KUKA KRL program: CONCERT.src, CONCERT.dat

--- CONCERT.src ---
&ACCESS RVO
&REL 519
&PARAM EDITMASK = *
&PARAM TEMPLATE = C:\KRC\Roboter\Template\vorgabe
&PARAM DISKPATH = KRC:\R1\Program\_KLAVIRISTA_V2\subprogram
DEF CONCERT( )
;FOLD INI
CONTINUE
IF NOT $ON_PATH THEN
  ;FOLD BASISTECH INI
    GLOBAL INTERRUPT DECL 3 WHEN $STOPMESS==TRUE DO IR_STOPM ( )
    INTERRUPT ON 3
    BAS (#INITMOV,0 )
  ;ENDFOLD (BASISTECH INI)
  ;FOLD USER INI
    ;Make your modifications here

  ;ENDFOLD (USER INI)
ENDIF
  ;ENDFOLD (INI)
;FOLD PTP HOME1 Vel=8 % PDAT5 ;%{PE}
;FOLD Parameters ;%{h}
;Params IlfProvider=kukaroboter.basistech.inlineforms.movement.old; Kuka.IsGlobalPoint=False; Kuka.PointName=HOME1; Kuka.BlendingEnabled=False; Kuka.MoveDataPtpName=PDAT5; Kuka.VelocityPtp=100; Kuka.CurrentCDSetIndex=0; Kuka.MovementParameterFieldEnabled=True; IlfCommand=PTP
;ENDFOLD
$BWDSTART = FALSE
PDAT_ACT = PPDAT5
FDAT_ACT = FHOME1
BAS(#PTP_PARAMS, 8)
SET_CD_PARAMS (0)
PTP XHOME1
;ENDFOLD

;FOLD PTP HOME1 Vel=8 % PDAT5 ;%{PE}
;FOLD Parameters ;%{h}
;Params IlfProvider=kukaroboter.basistech.inlineforms.movement.old; Kuka.IsGlobalPoint=False; Kuka.PointName=HOME1; Kuka.BlendingEnabled=False; Kuka.MoveDataPtpName=PDAT5; Kuka.VelocityPtp=100; Kuka.CurrentCDSetIndex=0; Kuka.MovementParameterFieldEnabled=True; IlfCommand=PTP
;ENDFOLD
$BWDSTART = FALSE
PDAT_ACT = PPDAT5
FDAT_ACT = FHOME1
BAS(#PTP_PARAMS, 8)
SET_CD_PARAMS (0)
PTP XHOME1
;ENDFOLD

END
GLOBAL DEF PLAY(KEY:IN, TIME:IN, HOLD:IN)
;FOLD Variables INI
REAL KEY
INT TIME
INT HOLD
INT PRESS
INT SPEED
REAL SHIFT
;ENDFOLD
PRESS = 10
SHIFT = 23.3
SPEED = 17
$TIMER_STOP[1]=FALSE
;FOLD STATUS TREATMENT
KEY = KEY+7
IF KEY < 11 THEN
XP1 = START4
ELSE
XP1 = START5
ENDIF
;IF KEY <= 8 THEN
;XP1 = START1
;ENDIF
;IF (KEY > 8) AND (KEY < 11) THEN
;XP1 = START2
;ENDIF
;IF KEY >= 11 THEN
;XP1 = START3
;ENDIF
;ENDFOLD

XP1.X = XP1.X + (KEY-1) * SHIFT
;FOLD PTP P1 Vel=100 % PDAT1 Tool[4]:TQGripper Base[1]:Piano ;%{PE}
;FOLD Parameters ;%{h}
;Params IlfProvider=kukaroboter.basistech.inlineforms.movement.old; Kuka.IsGlobalPoint=False; Kuka.PointName=P1; Kuka.BlendingEnabled=False; Kuka.MoveDataPtpName=PDAT1; Kuka.VelocityPtp=100; Kuka.CurrentCDSetIndex=0; Kuka.MovementParameterFieldEnabled=True; IlfCommand=PTP
;ENDFOLD
$BWDSTART = FALSE
PDAT_ACT = PPDAT1
FDAT_ACT = FP1
BAS(#PTP_PARAMS, SPEED)
SET_CD_PARAMS (0)
PTP XP1
;ENDFOLD
XP1.Z = XP1.Z - PRESS
WAIT FOR ($TIMER[1] > TIME)
;FOLD PTP P1 Vel=25 % PDAT1 Tool[4]:TQGripper Base[1]:Piano ;%{PE}
;FOLD Parameters ;%{h}
;Params IlfProvider=kukaroboter.basistech.inlineforms.movement.old; Kuka.IsGlobalPoint=False; Kuka.PointName=P1; Kuka.BlendingEnabled=True; Kuka.MoveDataPtpName=PDAT1; Kuka.VelocityPtp=100; Kuka.CurrentCDSetIndex=0; Kuka.MovementParameterFieldEnabled=True; IlfCommand=PTP
;ENDFOLD
$BWDSTART = FALSE
PDAT_ACT = PPDAT1
FDAT_ACT = FP1
BAS(#PTP_PARAMS, SPEED)
SET_CD_PARAMS (0)
PTP XP1
;ENDFOLD
$TIMER[1] = 0
XP1.Z = XP1.Z + PRESS
WAIT FOR ($TIMER[1] > HOLD)
;FOLD PTP P1 Vel=100 % PDAT1 Tool[4]:TQGripper Base[1]:Piano ;%{PE}
;FOLD Parameters ;%{h}
;Params IlfProvider=kukaroboter.basistech.inlineforms.movement.old; Kuka.IsGlobalPoint=False; Kuka.PointName=P1; Kuka.BlendingEnabled=True; Kuka.MoveDataPtpName=PDAT1; Kuka.VelocityPtp=100; Kuka.CurrentCDSetIndex=0; Kuka.MovementParameterFieldEnabled=True; IlfCommand=PTP
;ENDFOLD
$BWDSTART = FALSE
PDAT_ACT = PPDAT1
FDAT_ACT = FP1
BAS(#PTP_PARAMS, SPEED)
SET_CD_PARAMS (0)
PTP XP1
;ENDFOLD
$TIMER_STOP[1]=TRUE
$TIMER[1] = 0
RETURN
END
GLOBAL DEF FPLAY(KEY:IN, TIME:IN, HOLD:IN)
;FOLD Variables INI
INT KEY
INT TIME
INT HOLD
INT PRESS
INT SPEED
REAL SHIFT
;ENDFOLD
PRESS = 10
SHIFT = 23.3
SPEED = 17
;bylo to 25
$ADVANCE = 0
;FOLD STATUS TREATMENT
IF KEY < 11 THEN
XP2 = START4
ELSE
XP2 = START5
ENDIF
;ENDFOLD
;XP2=XP3
XP2.X = XP2.X + (KEY-1) * SHIFT
;FOLD PTP P2 Vel=100 % PDAT2 Tool[4]:TQGripper Base[1]:Piano ;%{PE}
;FOLD Parameters ;%{h}
;Params IlfProvider=kukaroboter.basistech.inlineforms.movement.old; Kuka.IsGlobalPoint=False; Kuka.PointName=P2; Kuka.BlendingEnabled=False; Kuka.MoveDataPtpName=PDAT2; Kuka.VelocityPtp=100; Kuka.CurrentCDSetIndex=0; Kuka.MovementParameterFieldEnabled=True; IlfCommand=PTP
;ENDFOLD
$BWDSTART = FALSE
PDAT_ACT = PPDAT2
FDAT_ACT = FP2
BAS(#PTP_PARAMS, SPEED)
SET_CD_PARAMS (0)
PTP XP2
;ENDFOLD
XP2.Z = XP2.Z - PRESS

$ADVANCE = 3
WAIT FOR ($TIMER[5] > TIME)
;$TIMER_STOP[3] = FALSE
;FOLD PTP P2 Vel=25 % PDAT2 Tool[4]:TQGripper Base[1]:Piano ;%{PE}
;FOLD Parameters ;%{h}
;Params IlfProvider=kukaroboter.basistech.inlineforms.movement.old; Kuka.IsGlobalPoint=False; Kuka.PointName=P2; Kuka.BlendingEnabled=True; Kuka.MoveDataPtpName=PDAT2; Kuka.VelocityPtp=100; Kuka.CurrentCDSetIndex=0; Kuka.MovementParameterFieldEnabled=True; IlfCommand=PTP
;ENDFOLD
$BWDSTART = FALSE
PDAT_ACT = PPDAT2
FDAT_ACT = FP2
BAS(#PTP_PARAMS, SPEED)
SET_CD_PARAMS (0)
PTP XP2
;ENDFOLD
;$TIMER_STOP[3] = TRUE
XP2.Z = XP2.Z + PRESS
WAIT FOR ($TIMER[5] > HOLD)
;FOLD PTP P2 Vel=100 % PDAT2 Tool[4]:TQGripper Base[1]:Piano ;%{PE}
;FOLD Parameters ;%{h}
;Params IlfProvider=kukaroboter.basistech.inlineforms.movement.old; Kuka.IsGlobalPoint=False; Kuka.PointName=P2; Kuka.BlendingEnabled=True; Kuka.MoveDataPtpName=PDAT2; Kuka.VelocityPtp=100; Kuka.CurrentCDSetIndex=0; Kuka.MovementParameterFieldEnabled=True; IlfCommand=PTP
;ENDFOLD
$BWDSTART = FALSE
PDAT_ACT = PPDAT2
FDAT_ACT = FP2
BAS(#PTP_PARAMS, SPEED)
SET_CD_PARAMS (0)
PTP XP2
;ENDFOLD

RETURN
END
GLOBAL DEF GRIPPER(STATE:IN,CEKEJ:IN)
INT STATE
BOOL CEKEJ

WAIT SEC 0

PULSE($OUT[1+STATE], TRUE, 0.75)
IF CEKEJ THEN
WAIT SEC 0.75
ENDIF
END

GLOBAL DEF PLAY_1(KEY:IN, TIME:IN, HOLD:IN)
;FOLD Variables INI
REAL KEY
INT TIME
INT HOLD
INT PRESS
INT SPEED
REAL SHIFT
;ENDFOLD
KEY=KEY/100
PRESS = 5
SHIFT = 36.3
SPEED = 17
$TIMER_STOP[1]=FALSE
;FOLD STATUS TREATMENT
KEY = KEY+7
IF KEY < 11 THEN
XP7 = START9
ELSE
XP7 = START10
ENDIF
;IF KEY <= 8 THEN
;XP7 = START1
;ENDIF
;IF (KEY > 8) AND (KEY < 11) THEN
;XP7 = START2
;ENDIF
;IF KEY >= 11 THEN
;XP7 = START3
;ENDIF
;ENDFOLD

XP7.X = XP7.X + (KEY-1) * SHIFT
;FOLD PTP P7 Vel=100 % PDAT9 Tool[4]:TQGripper Base[1]:Piano ;%{PE}
;FOLD Parameters ;%{h}
;Params IlfProvider=kukaroboter.basistech.inlineforms.movement.old; Kuka.IsGlobalPoint=False; Kuka.PointName=P7; Kuka.BlendingEnabled=False; Kuka.MoveDataPtpName=PDAT9; Kuka.VelocityPtp=100; Kuka.CurrentCDSetIndex=0; Kuka.MovementParameterFieldEnabled=True; IlfCommand=PTP
;ENDFOLD
$BWDSTART = FALSE
PDAT_ACT = PPDAT9
FDAT_ACT = FP7
BAS(#PTP_PARAMS, SPEED)
SET_CD_PARAMS (0)
PTP XP7
;ENDFOLD
XP7.Z = XP7.Z - (PRESS+6)
WAIT FOR ($TIMER[1] > TIME)
;FOLD PTP P7 Vel=25 % PDAT9 Tool[4]:TQGripper Base[1]:Piano ;%{PE}
;FOLD Parameters ;%{h}
;Params IlfProvider=kukaroboter.basistech.inlineforms.movement.old; Kuka.IsGlobalPoint=False; Kuka.PointName=P7; Kuka.BlendingEnabled=True; Kuka.MoveDataPtpName=PDAT9; Kuka.VelocityPtp=100; Kuka.CurrentCDSetIndex=0; Kuka.MovementParameterFieldEnabled=True; IlfCommand=PTP
;ENDFOLD
$BWDSTART = FALSE
PDAT_ACT = PPDAT9
FDAT_ACT = FP7
BAS(#PTP_PARAMS, SPEED)
SET_CD_PARAMS (0)
PTP XP7
;ENDFOLD
$TIMER[1] = 0
XP7.Y = XP7.Y - 40
;FOLD PTP P9 Vel=25 % PDAT10 Tool[4]:TQGripper Base[1]:Piano ;%{PE}
;FOLD Parameters ;%{h}
;Params IlfProvider=kukaroboter.basistech.inlineforms.movement.old; Kuka.IsGlobalPoint=False; Kuka.PointName=P9; Kuka.BlendingEnabled=True; Kuka.MoveDataPtpName=PDAT10; Kuka.VelocityPtp=100; Kuka.CurrentCDSetIndex=0; Kuka.MovementParameterFieldEnabled=True; IlfCommand=PTP
;ENDFOLD
$BWDSTART = FALSE
PDAT_ACT = PPDAT10
FDAT_ACT = FP8
BAS(#PTP_PARAMS, SPEED)
SET_CD_PARAMS (0)
PTP XP9
;ENDFOLD

XP7.Z = XP7.Z + PRESS
WAIT FOR ($TIMER[1] > HOLD)
;FOLD PTP P7 Vel=100 % PDAT9 Tool[4]:TQGripper Base[1]:Piano ;%{PE}
;FOLD Parameters ;%{h}
;Params IlfProvider=kukaroboter.basistech.inlineforms.movement.old; Kuka.IsGlobalPoint=False; Kuka.PointName=P7; Kuka.BlendingEnabled=True; Kuka.MoveDataPtpName=PDAT9; Kuka.VelocityPtp=100; Kuka.CurrentCDSetIndex=0; Kuka.MovementParameterFieldEnabled=True; IlfCommand=PTP
;ENDFOLD
$BWDSTART = FALSE
PDAT_ACT = PPDAT9
FDAT_ACT = FP7
BAS(#PTP_PARAMS, SPEED)
SET_CD_PARAMS (0)
PTP XP7
;ENDFOLD
$TIMER_STOP[1]=TRUE
$TIMER[1] = 0
RETURN
END

GLOBAL DEF PLAYRT(KEY:IN, TIME:IN)
  ;FOLD Variables INI
  REAL KEY
  INT TIME

  INT PRESS
  INT SPEED
  REAL SHIFT
  ;ENDFOLD
  PRESS = 10
  SHIFT = 23.3
  SPEED = 17
  $TIMER_STOP[1]=FALSE
  ;FOLD STATUS TREATMENT
  ;KEY = KEY
  IF KEY < 11 THEN
  XP1 = START4
  ELSE
  XP1 = START5
  ENDIF
  IF KEY <= 8 THEN
  XP1 = START1
  ENDIF
  IF (KEY > 8) AND (KEY < 11) THEN
  XP1 = START2
  ENDIF
  IF KEY >= 11 THEN
  XP1 = START3
  ENDIF
  ;ENDFOLD

  XP1.X = XP1.X + (KEY-1) * SHIFT
  ;FOLD PTP P1 Vel=100 % PDAT1 Tool[4]:TQGripper Base[1]:Piano ;%{PE}

  ;FOLD Parameters ;%{h}
  ;Params IlfProvider=kukaroboter.basistech.inlineforms.movement.old; Kuka.IsGlobalPoint=False; Kuka.PointName=P1; Kuka.BlendingEnabled=False; Kuka.MoveDataPtpName=PDAT1; Kuka.VelocityPtp=100; Kuka.CurrentCDSetIndex=0; Kuka.MovementParameterFieldEnabled=True; IlfCommand=PTP
  ;ENDFOLD
  $BWDSTART = FALSE
  PDAT_ACT = PPDAT1
  FDAT_ACT = FP1
  BAS(#PTP_PARAMS, SPEED)
  SET_CD_PARAMS (0)
  PTP XP1
  ;ENDFOLD
  XP1.Z = XP1.Z - PRESS
  WAIT FOR ($TIMER[1] > TIME)
  ;FOLD PTP P1 Vel=25 % PDAT1 Tool[4]:TQGripper Base[1]:Piano ;%{PE}
  ;FOLD Parameters ;%{h}
  ;Params IlfProvider=kukaroboter.basistech.inlineforms.movement.old; Kuka.IsGlobalPoint=False; Kuka.PointName=P1; Kuka.BlendingEnabled=True; Kuka.MoveDataPtpName=PDAT1; Kuka.VelocityPtp=100; Kuka.CurrentCDSetIndex=0; Kuka.MovementParameterFieldEnabled=True; IlfCommand=PTP
  ;ENDFOLD
  $BWDSTART = FALSE
  PDAT_ACT = PPDAT1
  FDAT_ACT = FP1
  BAS(#PTP_PARAMS, SPEED)
  SET_CD_PARAMS (0)
  PTP XP1
  ;ENDFOLD
  $TIMER[1] = 0
  XP1.Z = XP1.Z + PRESS
  WAIT FOR ($TIMER[1] > PyNoteDuration)
  ;FOLD PTP P1 Vel=100 % PDAT1 Tool[4]:TQGripper Base[1]:Piano ;%{PE}
  ;FOLD Parameters ;%{h}
  ;Params IlfProvider=kukaroboter.basistech.inlineforms.movement.old; Kuka.IsGlobalPoint=False; Kuka.PointName=P1; Kuka.BlendingEnabled=True; Kuka.MoveDataPtpName=PDAT1; Kuka.VelocityPtp=100; Kuka.CurrentCDSetIndex=0; Kuka.MovementParameterFieldEnabled=True; IlfCommand=PTP
  ;ENDFOLD
  $BWDSTART = FALSE
  PDAT_ACT = PPDAT1
  FDAT_ACT = FP1
  BAS(#PTP_PARAMS, SPEED)
  SET_CD_PARAMS (0)
  PTP XP1
  ;ENDFOLD
  $TIMER_STOP[1]=TRUE
  $TIMER[1] = 0
  PyGoToNote = -256
  RETURN
  END

--- CONCERT.dat ---
&ACCESS RVO
&REL 519
&PARAM EDITMASK = *
&PARAM TEMPLATE = C:\KRC\Roboter\Template\vorgabe
&PARAM DISKPATH = KRC:\R1\Program\_KLAVIRISTA_V2\subprogram
DEFDAT  CONCERT
;FOLD EXTERNAL DECLARATIONS;%{PE}%MKUKATPBASIS,%CEXT,%VCOMMON,%P
;FOLD BASISTECH EXT;%{PE}%MKUKATPBASIS,%CEXT,%VEXT,%P
EXT  BAS (BAS_COMMAND  :IN,REAL  :IN )
DECL INT TURN
;ENDFOLD (BASISTECH EXT)
;FOLD USER EXT;%{E}%MKUKATPUSER,%CEXT,%VEXT,%P
;Make your modifications here

;ENDFOLD (USER EXT)
;ENDFOLD (EXTERNAL DECLARATIONS)
DECL E6POS START1={X 16.7000,Y 25.0000,Z 20.0000,A 138.000,B 4.20000,C -173.300,S 2,T 10,E1 0.0,E2 0.0,E3 0.0,E4 0.0,E5 0.0,E6 0.0}
DECL E6POS START2={X 16.7000,Y 25.0000,Z 20.0000,A 138.000,B 4.20000,C -173.300,S 2,T 2,E1 0.0,E2 0.0,E3 0.0,E4 0.0,E5 0.0,E6 0.0}
DECL E6POS START3={X 16.7000,Y 25.0000,Z 20.0000,A 138.000,B 4.20000,C -173.300,S 2,T 3,E1 0.0,E2 0.0,E3 0.0,E4 0.0,E5 0.0,E6 0.0}
DECL E6POS XP1={X 307.250,Y 24.3000,Z 6.50000,A -85.0000,B 0.0,C 179.900,S 2,T 3,E1 0.0,E2 0.0,E3 0.0,E4 0.0,E5 0.0,E6 0.0}
DECL FDAT FP1={TOOL_NO 4,BASE_NO 1,IPO_FRAME #BASE,POINT2[] " "}
DECL PDAT PPDAT1={VEL 100.000,ACC 100.000,APO_DIST 500.000,APO_MODE #CDIS,GEAR_JERK 100.000,EXAX_IGN 0}
DECL PDAT PPDAT5={VEL 100.000,ACC 100.000,APO_DIST 500.000,APO_MODE #CDIS,GEAR_JERK 100.000,EXAX_IGN 0}
DECL FDAT FHOME1={TOOL_NO 3,BASE_NO 1,IPO_FRAME #BASE,POINT2[] " "}
DECL FDAT FHOME2={TOOL_NO 3,BASE_NO 1,IPO_FRAME #BASE,POINT2[] " "}
DECL PDAT PPDAT6={VEL 100.000,ACC 100.000,APO_DIST 500.000,APO_MODE #CDIS,GEAR_JERK 100.000,EXAX_IGN 0}
DECL FDAT FP2={TOOL_NO 4,BASE_NO 1,IPO_FRAME #BASE,POINT2[] " "}
DECL PDAT PPDAT2={VEL 100.000,ACC 100.000,APO_DIST 500.000,APO_MODE #CDIS,GEAR_JERK 100.000,EXAX_IGN 0}
DECL E6POS START6={X 16.7000,Y 25.0000,Z 20.0000,A 138.000,B 4.20000,C -173.300,S 2,T 3,E1 0.0,E2 0.0,E3 0.0,E4 0.0,E5 0.0,E6 0.0}
;;;
DECL E6POS START5={X 16.0000,Y 24.3000,Z 6.50000,A -85.0000,B 0.0,C 179.900,S 2,T 3,E1 0.0,E2 0.0,E3 0.0,E4 0.0,E5 0.0,E6 0.0}
DECL E6POS START4={X 16.0000,Y 24.3000,Z 6.50000,A -85.0000,B 0.0,C 179.900,S 2,T 2,E1 0.0,E2 0.0,E3 0.0,E4 0.0,E5 0.0,E6 0.0}
;;;
DECL E6POS XP2={X 551.899963,Y 24.3000,Z 6.50000,A -85.0000,B 0.0,C 179.900,S 2,T 3,E1 0.0,E2 0.0,E3 0.0,E4 0.0,E5 0.0,E6 0.0}
DECL MODULEPARAM_T LAST_TP_PARAMS={PARAMS[] "Kuka.PointName=P3; Kuka.FrameData.base_no=1; Kuka.FrameData.tool_no=4; Kuka.FrameData.ipo_frame=#BASE; Kuka.FrameData.point2=; Kuka.isglobalpoint=False; Kuka.MoveDataPtpName=PDAT3; Kuka.MovementDataPdat.apo_mode=#CDIS; Kuka.MovementDataPdat.apo_dist=500; Kuka.MovementData.vel=100; Kuka.MovementData.acc=100; Kuka.MovementData.exax_ign=0; Kuka.VelocityPtp=100; Kuka.BlendingEnabled=False; Kuka.APXEnabled=False; Kuka.CurrentCDSetIndex=0    "}
DECL E6POS XP3={X 17.2000,Y 24.3000,Z 5.00000,A -85.0000,B 0.0,C 179.900,S 2,T 2,E1 0.0,E2 0.0,E3 0.0,E4 0.0,E5 0.0,E6 0.0}
DECL FDAT FP3={TOOL_NO 4,BASE_NO 1,IPO_FRAME #BASE,POINT2[] " "}
DECL PDAT PPDAT3={VEL 100.000,ACC 100.000,APO_DIST 500.000,APO_MODE #CDIS,GEAR_JERK 100.000,EXAX_IGN 0}
DECL FDAT FP4={TOOL_NO 4,BASE_NO 1,IPO_FRAME #BASE,POINT2[] " "}
DECL PDAT PPDAT4={VEL 100.000,ACC 100.000,APO_DIST 500.000,APO_MODE #CDIS,GEAR_JERK 100.000,EXAX_IGN 0}
DECL E6POS START8={X 16.0000,Y 24.3000,Z 6.50000,A -85.0000,B 0.0,C 179.900,S 2,T 3,E1 0.0,E2 0.0,E3 0.0,E4 0.0,E5 0.0,E6 0.0}
DECL E6POS START7={X 16.0000,Y 24.3000,Z 6.50000,A -85.0000,B 0.0,C 179.900,S 2,T 2,E1 0.0,E2 0.0,E3 0.0,E4 0.0,E5 0.0,E6 0.0}
DECL E6POS XP4={X 307.250,Y 24.3000,Z 6.50000,A -85.0000,B 0.0,C 179.900,S 2,T 3,E1 0.0,E2 0.0,E3 0.0,E4 0.0,E5 0.0,E6 0.0}
DECL E6POS XP5={X 307.250,Y 24.3000,Z 6.50000,A -85.0000,B 0.0,C 179.900,S 2,T 3,E1 0.0,E2 0.0,E3 0.0,E4 0.0,E5 0.0,E6 0.0}
DECL FDAT FP5={TOOL_NO 4,BASE_NO 1,IPO_FRAME #BASE,POINT2[] " "}
DECL PDAT PPDAT7={VEL 100.000,ACC 100.000,APO_DIST 500.000,APO_MODE #CDIS,GEAR_JERK 100.000,EXAX_IGN 0}
DECL E6POS XP6={X 307.250,Y 24.3000,Z 6.50000,A -85.0000,B 0.0,C 179.900,S 2,T 3,E1 0.0,E2 0.0,E3 0.0,E4 0.0,E5 0.0,E6 0.0}
DECL FDAT FP6={TOOL_NO 4,BASE_NO 1,IPO_FRAME #BASE,POINT2[] " "}
DECL PDAT PPDAT8={VEL 100.000,ACC 100.000,APO_DIST 500.000,APO_MODE #CDIS,GEAR_JERK 100.000,EXAX_IGN 0}
DECL FDAT FP7={TOOL_NO 4,BASE_NO 1,IPO_FRAME #BASE,POINT2[] " "}
DECL PDAT PPDAT9={VEL 100.000,ACC 100.000,APO_DIST 500.000,APO_MODE #CDIS,GEAR_JERK 100.000,EXAX_IGN 0}
DECL E6POS START10={X 16.0000,Y 24.3000,Z 6.50000,A -85.0000,B 0.0,C 179.900,S 2,T 3,E1 0.0,E2 0.0,E3 0.0,E4 0.0,E5 0.0,E6 0.0}
DECL E6POS START9={X 16.0000,Y 24.3000,Z 6.50000,A -85.0000,B 0.0,C 179.900,S 2,T 2,E1 0.0,E2 0.0,E3 0.0,E4 0.0,E5 0.0,E6 0.0}
DECL E6POS XP7={X 270.099976,Y 24.3000,Z 6.50000,A -85.0000,B 0.0,C 179.900,S 2,T 2,E1 0.0,E2 0.0,E3 0.0,E4 0.0,E5 0.0,E6 0.0}
DECL E6POS XP9={X 307.250,Y 24.3000,Z 6.50000,A -85.0000,B 0.0,C 179.900,S 2,T 3,E1 0.0,E2 0.0,E3 0.0,E4 0.0,E5 0.0,E6 0.0}
DECL FDAT FP8={TOOL_NO 4,BASE_NO 1,IPO_FRAME #BASE,POINT2[] " "}
DECL PDAT PPDAT10={VEL 100.000,ACC 100.000,APO_DIST 500.000,APO_MODE #CDIS,GEAR_JERK 100.000,EXAX_IGN 0}
DECL E6POS XP8={X 307.250,Y 24.3000,Z 6.50000,A -85.0000,B 0.0,C 179.900,S 2,T 3,E1 0.0,E2 0.0,E3 0.0,E4 0.0,E5 0.0,E6 0.0}
ENDDAT
